{attribute 'qualified_only'}
VAR_GLOBAL
	var01		:	INT;
END_VAR

(* stored: Version 1.1.0.1, ProductVersion 3.1.4020.6
   GVL GVL01: Id {c5d628fc-f391-463e-af9c-f89978d6d7e0} *)
